{attribute 'GeneratedUsingTerminal: EP7047-1032-0021'}
{attribute addProperty BoxType "EP7047-1032-0021"}
{attribute addProperty Id "ENC_Status_compactAT %I*ENC_Status_compact_4D066E1A16STM_StatusAT %I*STM_Status_DE0D6B3712ENC_Control_compactAT %Q*ENC_Control_compact_21E2D14D6STM_ControlAT %Q*STM_Control_BA4CE3524STM_VelocityAT %Q*STM_Velocity_A47A3F412WcStateAT %I*WcState_9091E0EB2InfoDataAT %I*InfoData_3B4F4E8A4"}
{attribute addProperty CRC "3068540315"}
{attribute addProperty Size "46"}
TYPE EP7047_B6E6359B EXTENDS EtcSlaveTerminalBase_947E5A46 :
STRUCT
	{attribute addProperty Name "ENC_Status_compact"}
	ENC_Status_compact : ENC_Status_compact_4D066E1A;
	{attribute addProperty Name "STM_Status"}
	STM_Status : STM_Status_DE0D6B37;
	{attribute addProperty Name "ENC_Control_compact"}
	ENC_Control_compact : ENC_Control_compact_21E2D14D;
	{attribute addProperty Name "STM_Control"}
	STM_Control : STM_Control_BA4CE352;
	{attribute addProperty Name "STM_Velocity"}
	STM_Velocity : STM_Velocity_A47A3F41;
	{attribute addProperty Name "WcState"}
	WcState : WcState_9091E0EB;
	{attribute addProperty Name "InfoData"}
	InfoData : InfoData_3B4F4E8A;
END_STRUCT
END_TYPE

(* stored: Version 1.2.0.0, ProductVersion 3.1.4024.9
   DUT EP7047_B6E6359B: Id {16b2fdd9-b8b4-4659-832c-dae5b60bf2e7} *)
